# EPICS autosave request: basleracA130075gmApp/Db/plugin_settings.req
file "NDROI_settings.req",          P=$(PREFIX),  R=ROI1
file "NDStats_settings.req",        P=$(PREFIX),  R=Stats1
file "NDStats_settings.req",        P=$(PREFIX),  R=Stats2
file "NDTransform_settings.req",    P=$(PREFIX),  R=Transf1
